# EPICS autosave request: APD-ACE/apd-ace_settings.req
$(P):INTTIME
$(P):NREP
